FUNCTION_BLOCK Machine
  (* Version 1.0, 2006-11-02, Goran Cengic, Chalmers *)
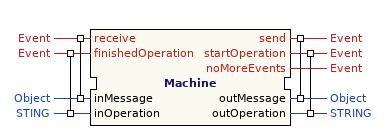
  EVENT_INPUT
    receive WITH inMessage;
    finishedOperation WITH inOperation;
  END_EVENT
  EVENT_OUTPUT
    send WITH outMessage;
    startOperation WITH outOperation;
    noMoreEvents;
  END_EVENT
  VAR_INPUT
    inMessage : Object;
    inOperation : STING;
  END_VAR
  VAR_OUTPUT
    outMessage : Object;
    outOperation : STRING;
  END_VAR
END_FUNCTION_BLOCK
